(* CODESYS project RTON.xml

Project tree, tasks and I/O mapping:
  function block RTON [LD]
*)

// RTON
FUNCTION_BLOCK RTON // Rententive Timer On
VAR_INPUT
	IN: BOOL; // Enable input bit.
	PT: TIME; // Preset time.
	Reset: BOOL; // Reset input bit.
END_VAR
VAR_OUTPUT
	Q: BOOL; // Output bit.
	ET: TIME; // Elapsed time.
END_VAR
VAR
	Timer: TON;
	FallingTrigger: F_TRIG;
	RisingTrigger: R_TRIG;
	RemainingTime: TIME;
	CurrentTime: TIME;
	TimeReset: BOOL;
END_VAR
VAR // added by the converter: edge detectors and wires of the graphical bodies
    _w1, _w2 : BOOL;
END_VAR

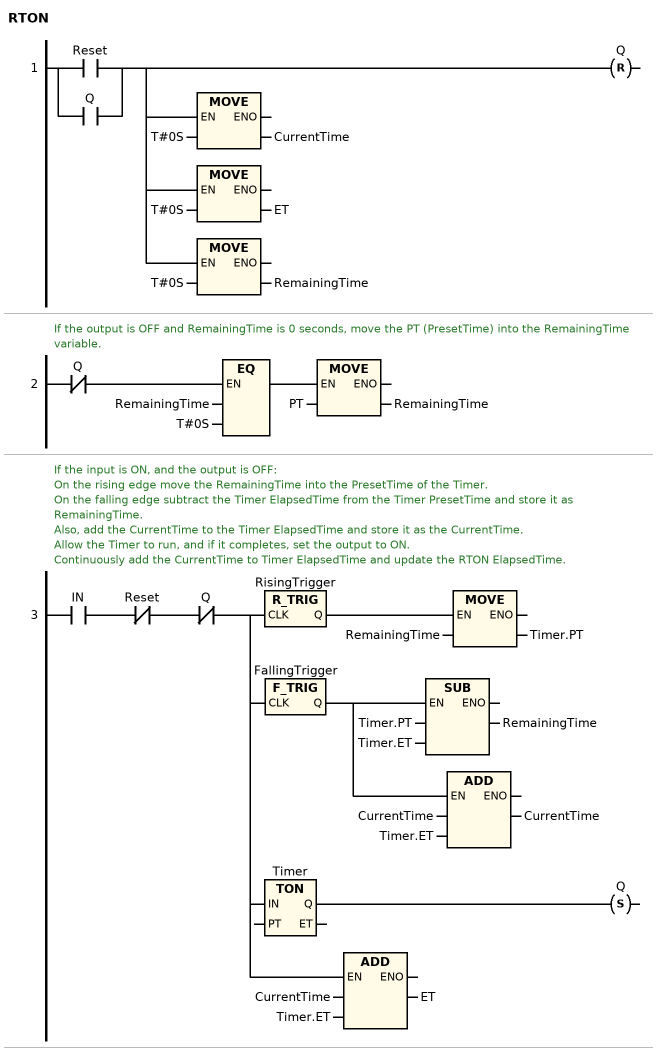
// NETWORK 1
_w1 := Reset OR Q;
Q R= _w1;
IF _w1 THEN CurrentTime := T#0S; END_IF
IF _w1 THEN ET := T#0S; END_IF
IF _w1 THEN RemainingTime := T#0S; END_IF

// NETWORK 2
// If the output is OFF and RemainingTime is 0 seconds, move the PT (PresetTime) into the RemainingTime variable.
IF NOT Q AND RemainingTime = T#0S THEN RemainingTime := PT; END_IF

// NETWORK 3
// If the input is ON, and the output is OFF:
//   On the rising edge move the RemainingTime into the PresetTime of the Timer.
//   On the falling edge subtract the Timer ElapsedTime from the Timer PresetTime and store it as RemainingTime.
//     Also, add the CurrentTime to the Timer ElapsedTime and store it as the CurrentTime.
//   Allow the Timer to run, and if it completes, set the output to ON.
//   Continuously add the CurrentTime to Timer ElapsedTime and update the RTON ElapsedTime.
_w2 := IN AND NOT Reset AND NOT Q;
RisingTrigger(CLK := _w2); // R_TRIG
IF RisingTrigger.Q THEN Timer.PT := RemainingTime; END_IF
FallingTrigger(CLK := _w2); // F_TRIG
IF FallingTrigger.Q THEN RemainingTime := Timer.PT - Timer.ET; END_IF
IF FallingTrigger.Q THEN CurrentTime := CurrentTime + Timer.ET; END_IF
Timer(IN := _w2); // TON
Q S= Timer.Q;
IF _w2 THEN ET := CurrentTime + Timer.ET; END_IF

END_FUNCTION_BLOCK
